FUNCTION_BLOCK FlashControl (* Flash Control Block Type *)
  (* Standard: 61499-2 *)
  (* Version 0.3, 2009-09-15, JHC, Holobloc Inc, Changed transition priorities. *)
  (* Version 0.2, 2003-12-04, JHC, Rockwell Automation, Renamed for better indexing. *)
  (* Version 0.1, 2002-11-05, JHC, Rockwell Automation, Corrected missing ST element in Algorithm REQ. *)
  (* Version 0.0, 2000-05-30, JHC, Rockwell Automation *)
  (* Compiler header: package fb.rt.template; *)
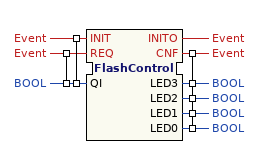
  EVENT_INPUT
    INIT WITH QI; (* Initialization Request *)
    REQ WITH QI; (* Normal Execution Request *)
  END_EVENT
  EVENT_OUTPUT
    INITO; (* Initialization Confirm *)
    CNF WITH LED3, LED2, LED1, LED0; (* Execution Confirmation *)
  END_EVENT
  VAR_INPUT
    QI : BOOL; (* Input event qualifier *)
  END_VAR
  VAR_OUTPUT
    LED3 : BOOL;
    LED2 : BOOL;
    LED1 : BOOL;
    LED0 : BOOL;
  END_VAR
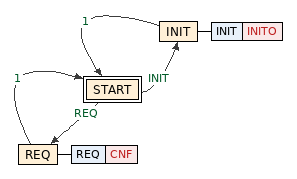
  EC_STATES
    START; (* Initial State *)
    INIT : INIT -> INITO; (* Initialization *)
    REQ : REQ -> CNF; (* Normal execution *)
  END_STATES
  EC_TRANSITIONS
    INIT TO START := 1;
    START TO REQ := REQ;
    START TO INIT := INIT;
    REQ TO START := 1;
  END_TRANSITIONS
  ALGORITHM INIT IN ST: (* Initialization algorithm *)
IF QI THEN
	LED0:=FALSE;
	LED1:=FALSE;
	LED2:=FALSE;
    LED3:=FALSE;
END_IF;
  END_ALGORITHM
  ALGORITHM REQ IN ST: (* Normally executed algorithm *)
LED0:=NOT LED0;
LED1:=NOT LED1;
LED2:=NOT LED2;
LED3:=NOT LED3;
  END_ALGORITHM
END_FUNCTION_BLOCK
